// Implicitly generated code : DO NOT EDIT
FUNCTION CheckDivLReal : LREAL
VAR_INPUT
	divisor:LREAL;
END_VAR

// Implicitly generated code : Only an Implementation suggestion
{noflow}
IF divisor = 0 THEN
	CheckDivLReal:=1;
ELSE
	CheckDivLReal:=divisor;
END_IF;
{flow}

END_FUNCTION

(* stored: Version 1.1.0.1, ProductVersion 3.1.4024.11
   POU CheckDivLReal: Id {c1073d60-fe93-4b53-b9c2-cb53eb68541d}, SpecialFunc CheckDivReal64 *)
